TYPE "FRK_TestRow"
VERSION : 0.1
   STRUCT
      CaseId : Int;
      Pass : Bool;
      Expected : DInt;
      Actual : DInt;
   END_STRUCT;

END_TYPE
